Fanuc KAREL source: IO0012.KL

-- PROVISIONAL review KL for V940-1; original PC SHA256 d50221fc37c102e4e688d8ed5e46ecfca3261178fc2c8c6133a8db39108f1475
-- Incomplete behavior may be omitted. Consult companion uncertainty JSON. Do not deploy.
PROGRAM IO0012
%NOLOCKGROUP
-- UNRESOLVED_LOCAL_POOL 5 cells at code offset 13; source declarations unknown
-- DIRECT_LOCAL_WORD_ACCESS alone does not prove INTEGER, REAL, or BOOLEAN
BEGIN
  -- V9_ZERO_TABLE_METADATA_HINT layout=0001; no indexed target words; source/name/runtime held
  -- V9_ZERO_GLOBAL_LAYOUT_HINT count-one $GROUP table, zero relocation slots, two routine descriptors; executable preamble and source held
  -- UNRESOLVED_PC offsets 0-18; opcodes 2B,2C,7B
  -- UNRESOLVED_PC offsets 23-30; opcodes 9D,23
  -- UNRESOLVED_PC offsets 35-49; opcodes 2E,22,9D,33,35
  -- UNRESOLVED_PC offsets 54-61; opcodes 9D,23
  -- UNRESOLVED_PC offsets 66-77; opcodes 2E,23
  -- UNRESOLVED_PC offsets 82-100; opcodes 03,21,9D,52,1B,9D,12,13,04,14
  -- UNRESOLVED_PC offsets 105-109; opcodes 7F
  -- UNRESOLVED_PC offsets 114-118; opcodes 27,AA
  -- UNRESOLVED_PC offsets 123-127; opcodes 7F
END IO0012
